(* Logix 5000 project; controller ERT303_BaseConfig vendor 1 type 14 code 226 rev 33.11; software revision 33.02 *)

TASK MainTask (continuous, watchdog 500 ms) : MainProgram
TASK SafetyTask (periodic, rate 20 ms, priority 10, watchdog 20 ms, safety) : SafetyProgram

MODULES
   Local : vendor 1 type 14 code 226 (5069 0, rev 33.11)
END_MODULES

TYPE _Blade :
STRUCT
   Raise : _sol_motion;
   Lower : _sol_motion;
END_STRUCT
END_TYPE

TYPE _clamp :
STRUCT
   Raise : _sol_motion;
   Lower : _sol_motion;
   Clamp : _sol_motion;
   Unclamp : _sol_motion;
END_STRUCT
END_TYPE

TYPE _Gantry :
STRUCT
   Adv_Z : _sol_motion;
   Ret_Z : _sol_motion;
   Adv_X : _sol_motion;
   Ret_X : _sol_motion;
   Grip : _sol_motion;
   Ungrip : _sol_motion;
   Adv_Y : _sol_motion;
   Ret_Y : _sol_motion;
END_STRUCT
END_TYPE

TYPE _modes :
STRUCT
   Auto : BOOL;   // Auto Mode
   Manual : BOOL;   // Manual Mode
   AutoCycle : BOOL;   // In Auto Cycle
END_STRUCT
END_TYPE

TYPE _motor :
STRUCT
   OkToMove : BOOL;   // Clear And OK To Move
   AutoCondition : BOOL;   // Auto Move Conditions Met
   Command : BOOL;   // Move Command
END_STRUCT
END_TYPE

TYPE _pusher :
STRUCT
   Adv : _sol_motion;   // Extend
   Ret : _sol_motion;   // Retract
END_STRUCT
END_TYPE

TYPE _sol_motion :
STRUCT
   OkToMove : BOOL;   // Clear And OK To Move
   AutoCondition : BOOL;   // Auto Move Conditions Met
   Command : BOOL;   // Move Command
   PosFdbk : BOOL;   // In Position Feedback
   Complete : BOOL;   // Motion Complete
   CompleteDelayTimer : TIMER;   // Motion Complete Delay Timer
   SlowFltTimer : TIMER;   // Slow Motion Fault Timer
   SlowFlt : BOOL;   // Slow Motion Fault
   SwitchFlt : BOOL;   // Switch Fault
END_STRUCT
END_TYPE

VAR_GLOBAL   (* controller tags *)
   AlarmSta1 : ALIAS FOR BOOL_OUT_17;   // ALARM AT STATION 1
   AlarmSta2 : ALIAS FOR BOOL_OUT_32;   // ALARM AT STATION 2
   BELT0 : ALIAS FOR BOOL_OUT_1;
   BELT1 : ALIAS FOR BOOL_OUT_2;
   BELT10 : ALIAS FOR BOOL_OUT_11;
   BELT11 : ALIAS FOR BOOL_OUT_12;
   BELT12 : ALIAS FOR BOOL_OUT_13;
   BELT13 : ALIAS FOR BOOL_OUT_14;
   BELT14 : ALIAS FOR BOOL_OUT_15;
   BELT2 : ALIAS FOR BOOL_OUT_3;
   BELT3 : ALIAS FOR BOOL_OUT_4;
   BELT4 : ALIAS FOR BOOL_OUT_5;
   BELT5 : ALIAS FOR BOOL_OUT_6;
   BELT6 : ALIAS FOR BOOL_OUT_7;
   BELT7 : ALIAS FOR BOOL_OUT_8;
   BELT8 : ALIAS FOR BOOL_OUT_9;
   BELT9 : ALIAS FOR BOOL_OUT_10;
   BELTWEIGHTSCALE : ALIAS FOR BOOL_OUT_16;
   BOOL_IN_1 : BOOL := 1;
   BOOL_IN_10 : BOOL;
   BOOL_IN_11 : BOOL;
   BOOL_IN_12 : BOOL;
   BOOL_IN_13 : BOOL;
   BOOL_IN_14 : BOOL;
   BOOL_IN_15 : BOOL;
   BOOL_IN_16 : BOOL;
   BOOL_IN_17 : BOOL;
   BOOL_IN_18 : BOOL;
   BOOL_IN_19 : BOOL;
   BOOL_IN_2 : BOOL;
   BOOL_IN_20 : BOOL;
   BOOL_IN_21 : BOOL;
   BOOL_IN_22 : BOOL;
   BOOL_IN_23 : BOOL;
   BOOL_IN_24 : BOOL;
   BOOL_IN_25 : BOOL;
   BOOL_IN_26 : BOOL;
   BOOL_IN_27 : BOOL;
   BOOL_IN_28 : BOOL;
   BOOL_IN_29 : BOOL;
   BOOL_IN_3 : BOOL := 1;
   BOOL_IN_30 : BOOL;
   BOOL_IN_31 : BOOL;
   BOOL_IN_32 : BOOL;
   BOOL_IN_33 : BOOL;
   BOOL_IN_34 : BOOL;
   BOOL_IN_35 : BOOL;
   BOOL_IN_36 : BOOL;
   BOOL_IN_4 : BOOL;
   BOOL_IN_5 : BOOL;
   BOOL_IN_6 : BOOL;
   BOOL_IN_7 : BOOL;
   BOOL_IN_8 : BOOL;
   BOOL_IN_9 : BOOL;
   BOOL_OUT_1 : BOOL;
   BOOL_OUT_10 : BOOL;
   BOOL_OUT_11 : BOOL;
   BOOL_OUT_12 : BOOL;
   BOOL_OUT_13 : BOOL;
   BOOL_OUT_14 : BOOL;
   BOOL_OUT_15 : BOOL;
   BOOL_OUT_16 : BOOL;
   BOOL_OUT_17 : BOOL := 1;
   BOOL_OUT_18 : BOOL;
   BOOL_OUT_19 : BOOL;
   BOOL_OUT_2 : BOOL;
   BOOL_OUT_20 : BOOL;
   BOOL_OUT_21 : BOOL;
   BOOL_OUT_22 : BOOL;
   BOOL_OUT_23 : BOOL;
   BOOL_OUT_24 : BOOL;
   BOOL_OUT_25 : BOOL;
   BOOL_OUT_26 : BOOL;
   BOOL_OUT_27 : BOOL;
   BOOL_OUT_28 : BOOL;
   BOOL_OUT_29 : BOOL := 1;
   BOOL_OUT_3 : BOOL;
   BOOL_OUT_30 : BOOL;
   BOOL_OUT_31 : BOOL := 1;
   BOOL_OUT_32 : BOOL := 1;
   BOOL_OUT_33 : BOOL;
   BOOL_OUT_34 : BOOL := 1;
   BOOL_OUT_35 : BOOL;
   BOOL_OUT_36 : BOOL;
   BOOL_OUT_37 : BOOL := 1;
   BOOL_OUT_38 : BOOL := 1;
   BOOL_OUT_39 : BOOL := 1;
   BOOL_OUT_4 : BOOL;
   BOOL_OUT_40 : BOOL := 1;
   BOOL_OUT_41 : BOOL;
   BOOL_OUT_42 : BOOL := 1;
   BOOL_OUT_43 : BOOL := 1;
   BOOL_OUT_44 : BOOL;
   BOOL_OUT_5 : BOOL;
   BOOL_OUT_6 : BOOL;
   BOOL_OUT_7 : BOOL;
   BOOL_OUT_8 : BOOL;
   BOOL_OUT_9 : BOOL;
   CURVEBELT0 : ALIAS FOR BOOL_OUT_18;
   CURVEBELT1 : ALIAS FOR BOOL_OUT_22;
   CURVEBELT2 : ALIAS FOR BOOL_OUT_19;
   CURVEBELT3 : ALIAS FOR BOOL_OUT_20;
   CURVEBELT4 : ALIAS FOR BOOL_OUT_21;
   DISPLAY0 : ALIAS FOR FLOAT_OUT_1;   // WEIGHT DISPLAY
   DISPLAY1 : ALIAS FOR INT_OUT_1;   // SHOWS TOTAL PARTS ON FRAGILE LINE
   DISPLAY2 : ALIAS FOR INT_OUT_2;   // SHOWS TOTAL NUMBER OF PARTS HANDLE BY SYSTEM
   EmergencyStop : ALIAS FOR BOOL_IN_1;   // EMERGENCY STOP BUTTON
   FactoryIOReset : ALIAS FOR BOOL_OUT_43;   // RESET BUTTON FOR WHOLE SYSTEM
   FLOAT_IN_1 : REAL;
   FLOAT_IN_10 : REAL;
   FLOAT_IN_11 : REAL;
   FLOAT_IN_12 : REAL;
   FLOAT_IN_2 : REAL;
   FLOAT_IN_3 : REAL;
   FLOAT_IN_4 : REAL;
   FLOAT_IN_5 : REAL;
   FLOAT_IN_6 : REAL;
   FLOAT_IN_7 : REAL;
   FLOAT_IN_8 : REAL;
   FLOAT_IN_9 : REAL;
   FLOAT_OUT_1 : REAL;
   FLOAT_OUT_10 : REAL;
   FLOAT_OUT_11 : REAL;
   FLOAT_OUT_12 : REAL;
   FLOAT_OUT_2 : REAL;
   FLOAT_OUT_3 : REAL;
   FLOAT_OUT_4 : REAL;
   FLOAT_OUT_5 : REAL;
   FLOAT_OUT_6 : REAL;
   FLOAT_OUT_7 : REAL;
   FLOAT_OUT_8 : REAL;
   FLOAT_OUT_9 : REAL;
   FRAGILESENSOR : ALIAS FOR BOOL_IN_5;   // SENSOR FOR FRAGILE PART COUNT AT STARTING OF FRAGILE LINE
   FRAGILESENSOR2 : ALIAS FOR BOOL_IN_23;   // SENSOR FOR FRAGILE PART COUNT AT ENDING OF FRAGILE LINE
   INT_IN_1 : DINT;
   INT_IN_10 : DINT;
   INT_IN_11 : DINT;
   INT_IN_12 : DINT;
   INT_IN_13 : DINT;
   INT_IN_14 : DINT;
   INT_IN_15 : DINT;
   INT_IN_16 : DINT;
   INT_IN_17 : DINT;
   INT_IN_18 : DINT;
   INT_IN_2 : DINT;
   INT_IN_3 : DINT;
   INT_IN_4 : DINT;
   INT_IN_5 : DINT;
   INT_IN_6 : DINT;
   INT_IN_7 : DINT;
   INT_IN_8 : DINT;
   INT_IN_9 : DINT;
   INT_OUT_1 : DINT := 3;
   INT_OUT_10 : DINT;
   INT_OUT_11 : DINT;
   INT_OUT_12 : DINT;
   INT_OUT_13 : DINT;
   INT_OUT_14 : DINT;
   INT_OUT_15 : DINT;
   INT_OUT_16 : DINT;
   INT_OUT_17 : DINT;
   INT_OUT_18 : DINT;
   INT_OUT_2 : DINT;
   INT_OUT_3 : DINT;
   INT_OUT_4 : DINT;
   INT_OUT_5 : DINT;
   INT_OUT_6 : DINT;
   INT_OUT_7 : DINT;
   INT_OUT_8 : DINT;
   INT_OUT_9 : DINT;
   PBRESET1 : ALIAS FOR BOOL_IN_16;   // RESET PB FOR STATION 1
   PBRESET2 : ALIAS FOR BOOL_IN_17;   // RESET PB OF STATION 2
   PIVOTARM0 : ALIAS FOR BOOL_OUT_23;   // MAIN PIVOT ARM
   PIVOTARM1 : ALIAS FOR BOOL_OUT_24;   // PIVOT ARM FOR SORTING OF BLUE PART
   PIVOTARM2 : ALIAS FOR BOOL_OUT_25;   // PIVOT ARM FOR SORTING OF GREEN PART
   PIVOTARMBELT0 : ALIAS FOR BOOL_OUT_26;
   PIVOTARMBELT1 : ALIAS FOR BOOL_OUT_27;
   PIVOTARMBELT2 : ALIAS FOR BOOL_OUT_28;
   SAFTEYDOOR : ALIAS FOR BOOL_IN_18;   // SAFTEYDOOR CONTROL
   STACKLTGREEN : ALIAS FOR BOOL_OUT_36;   // GREEN STACK LIGHT AT FRONT STATION
   STACKLTGREEN1 : ALIAS FOR BOOL_OUT_30;   // GREEN STACK LIGHT AT STATION 1
   STACKLTGREEN2 : ALIAS FOR BOOL_OUT_41;   // GREEN STACK LIGHT AT STATION 2
   STACKLTRED : ALIAS FOR BOOL_OUT_35;
   STACKLTRED1 : ALIAS FOR BOOL_OUT_29;   // RED STACK LIGHT AT STATION 1
   STACKLTRED2 : ALIAS FOR BOOL_OUT_40;   // RED STACK LIGHT AT STATION 2
   STACKLTYELLOW : ALIAS FOR BOOL_OUT_37;   // YELLOW STACK LIGHT AT FRONT
   STACKLTYELLOW1 : ALIAS FOR BOOL_OUT_31;   // YELLOW STACK LIGHT AT STATION 1
   STACKLTYELLOW2 : ALIAS FOR BOOL_OUT_42;   // YELLOW STACK LIGHT AT STATION 2
   STARTLT : ALIAS FOR BOOL_OUT_33;   // GREEN LIGHT OF START PB
   StartPB : ALIAS FOR BOOL_IN_2;   // START PUSH BUTTON
   STOPLT : ALIAS FOR BOOL_OUT_34;   // RED LIGHT OF STOP PB
   StopPB : ALIAS FOR BOOL_IN_3;   // STOP PUSH BUTTON
   VISION1A : ALIAS FOR BOOL_IN_6;
   VISION1B : ALIAS FOR BOOL_IN_7;
   VISION1C : ALIAS FOR BOOL_IN_8;
   VISION2A : ALIAS FOR BOOL_IN_9;
   VISION2B : ALIAS FOR BOOL_IN_10;
   VISION2C : ALIAS FOR BOOL_IN_11;
   VISION3A : ALIAS FOR BOOL_IN_12;
   VISION3B : ALIAS FOR BOOL_IN_13;
   VISION3C : ALIAS FOR BOOL_IN_14;
   VISION3D : ALIAS FOR BOOL_IN_15;
   VISION4A : ALIAS FOR BOOL_IN_19;
   VISION4B : ALIAS FOR BOOL_IN_20;
   VISION4C : ALIAS FOR BOOL_IN_21;
   VISION4D : ALIAS FOR BOOL_IN_22;
   WARNLTST1 : ALIAS FOR BOOL_OUT_39;   // WARN LIGHT AT FRAGILE PART PICKUP STATION
   WARNLTSTAIR : ALIAS FOR BOOL_OUT_38;   // WARN SIGNAL LIGHT AT STAIR
   WeightScale : ALIAS FOR FLOAT_IN_1;   // ACTUAL WEIGHT MEASURE AT WEIGHT SCALE
   WeightSensor : ALIAS FOR BOOL_IN_4;   // SENSOR AT WEIGHT SCALE
END_VAR

PROGRAM MainProgram   (* main routine MainRoutine *)
VAR
   ActualWeight : REAL;
   AllConveyorsRun : BOOL;   // All Conveyors present
   DelayTimer : TIMER := (PRE := 5000);   // DELAY OF 5 SECONDS AT WEIGHT BELT
   FRAGILEPARTS : COUNTER;
   FRAGILEPARTSTART : COUNTER := (ACC := 29, DN := 1);   // COUNTER OF FRAGILE PART AT START OF FRAGILE LINE
   FRAGILEPARTSTOP : COUNTER := (ACC := 26, DN := 1);   // COUNTER OF FRAGILE PART AT END OF FRAGILE LINE
   Partdelaycomplete : BOOL;   // PART DELAY COMPLETION
   TotalParts : COUNTER;   // TOTAL PARTS HANDLE BY SYSTEM
END_VAR

ROUTINE CONVEYOR_SYSTEM   (* ladder *)
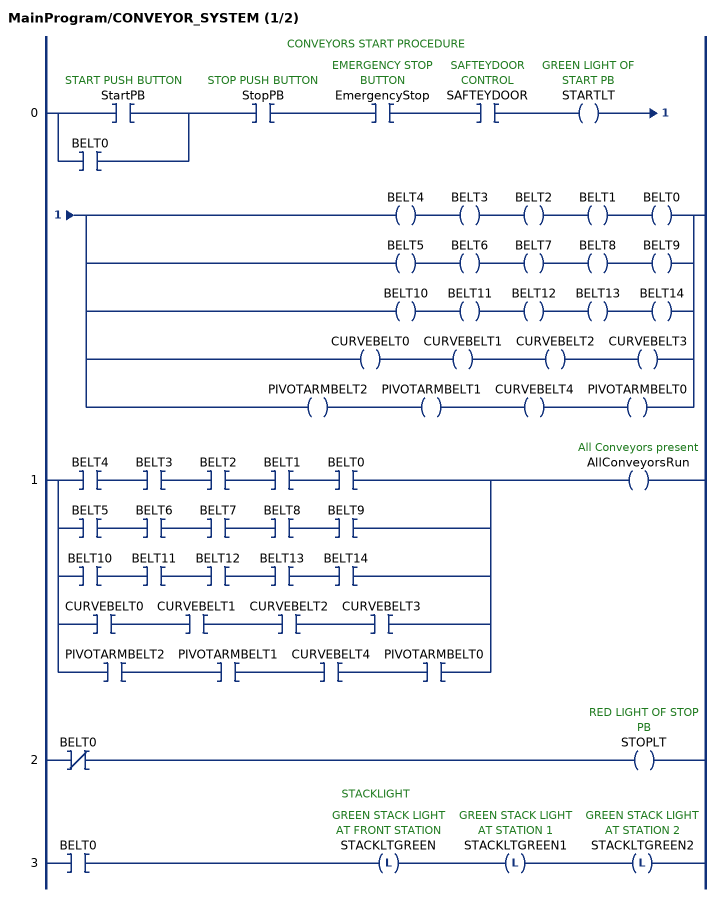
   // CONVEYORS START PROCEDURE
   0: [XIC(StartPB) ,XIC(BELT0) ]XIC(StopPB)XIC(EmergencyStop)XIC(SAFTEYDOOR)OTE(STARTLT)[OTE(BELT4) OTE(BELT3) OTE(BELT2) OTE(BELT1) OTE(BELT0) ,OTE(BELT5) OTE(BELT6) OTE(BELT7) OTE(BELT8) OTE(BELT9) ,OTE(BELT10) OTE(BELT11) OTE(BELT12) OTE(BELT13) OTE(BELT14) ,OTE(CURVEBELT0) OTE(CURVEBELT1) OTE(CURVEBELT2) OTE(CURVEBELT3) ,OTE(PIVOTARMBELT2) OTE(PIVOTARMBELT1) OTE(CURVEBELT4) OTE(PIVOTARMBELT0) ];
   1: [XIC(BELT4) XIC(BELT3) XIC(BELT2) XIC(BELT1) XIC(BELT0) ,XIC(BELT5) XIC(BELT6) XIC(BELT7) XIC(BELT8) XIC(BELT9) ,XIC(BELT10) XIC(BELT11) XIC(BELT12) XIC(BELT13) XIC(BELT14) ,XIC(CURVEBELT0) XIC(CURVEBELT1) XIC(CURVEBELT2) XIC(CURVEBELT3) ,XIC(PIVOTARMBELT2) XIC(PIVOTARMBELT1) XIC(CURVEBELT4) XIC(PIVOTARMBELT0) ]OTE(AllConveyorsRun);
   2: XIO(BELT0)OTE(STOPLT);
   // STACKLIGHT
   3: XIC(BELT0)OTL(STACKLTGREEN)OTL(STACKLTGREEN1)OTL(STACKLTGREEN2);
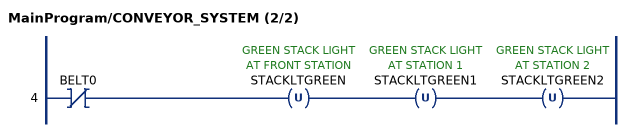
   4: XIO(BELT0)OTU(STACKLTGREEN)OTU(STACKLTGREEN1)OTU(STACKLTGREEN2);
END_ROUTINE

ROUTINE LIGHTING   (* ladder *)
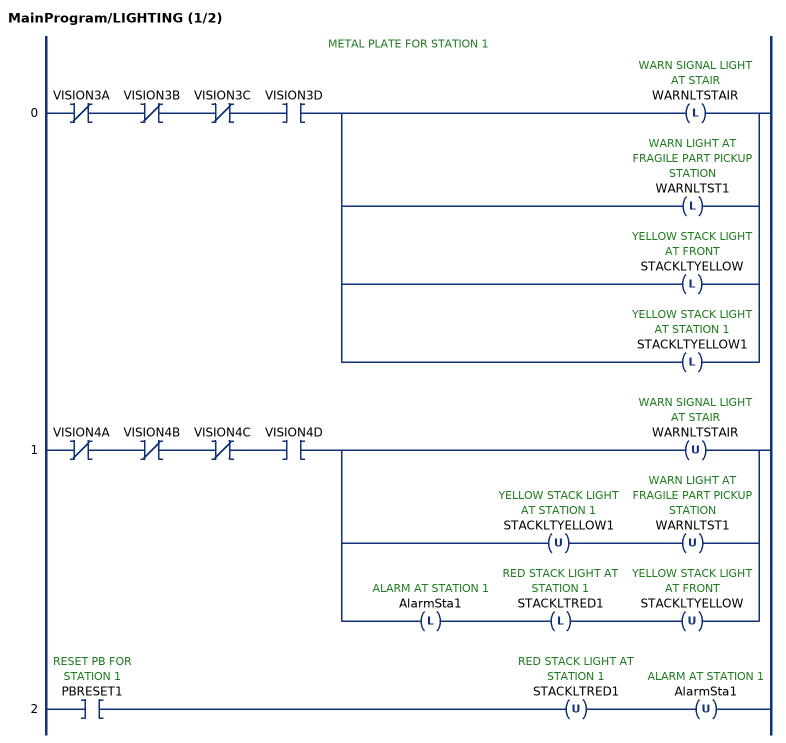
   // METAL PLATE FOR STATION 1
   0: XIO(VISION3A)XIO(VISION3B)XIO(VISION3C)XIC(VISION3D)[OTL(WARNLTSTAIR) ,OTL(WARNLTST1) ,OTL(STACKLTYELLOW) ,OTL(STACKLTYELLOW1) ];
   1: XIO(VISION4A)XIO(VISION4B)XIO(VISION4C)XIC(VISION4D)[OTU(WARNLTSTAIR) ,OTU(STACKLTYELLOW1) OTU(WARNLTST1) ,OTL(AlarmSta1) OTL(STACKLTRED1) OTU(STACKLTYELLOW) ];
   2: XIC(PBRESET1)OTU(STACKLTRED1)OTU(AlarmSta1);
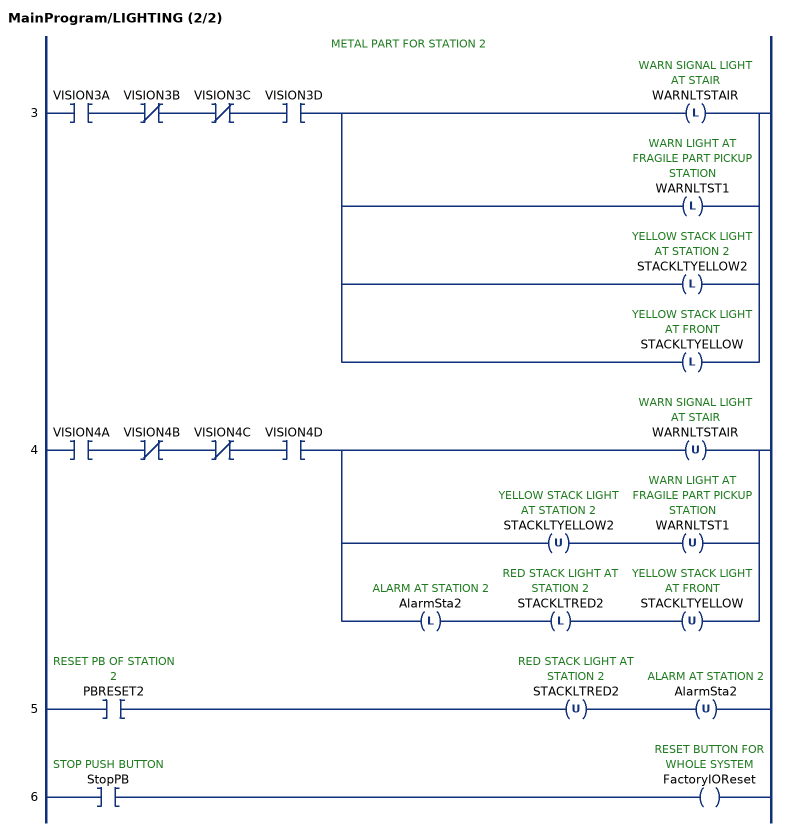
   // METAL PART FOR STATION 2
   3: XIC(VISION3A)XIO(VISION3B)XIO(VISION3C)XIC(VISION3D)[OTL(WARNLTSTAIR) ,OTL(WARNLTST1) ,OTL(STACKLTYELLOW2) ,OTL(STACKLTYELLOW) ];
   4: XIC(VISION4A)XIO(VISION4B)XIO(VISION4C)XIC(VISION4D)[OTU(WARNLTSTAIR) ,OTU(STACKLTYELLOW2) OTU(WARNLTST1) ,OTL(AlarmSta2) OTL(STACKLTRED2) OTU(STACKLTYELLOW) ];
   5: XIC(PBRESET2)OTU(STACKLTRED2)OTU(AlarmSta2);
   6: XIC(StopPB)OTE(FactoryIOReset);
END_ROUTINE

ROUTINE MainRoutine   (* ladder *)
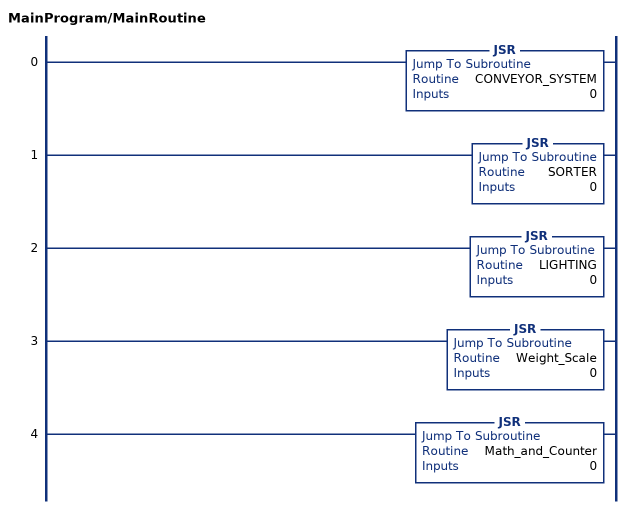
   0: JSR(CONVEYOR_SYSTEM,0);
   1: JSR(SORTER,0);
   2: JSR(LIGHTING,0);
   3: JSR(Weight_Scale,0);
   4: JSR(Math_and_Counter,0);
END_ROUTINE

ROUTINE Math_and_Counter   (* ladder *)
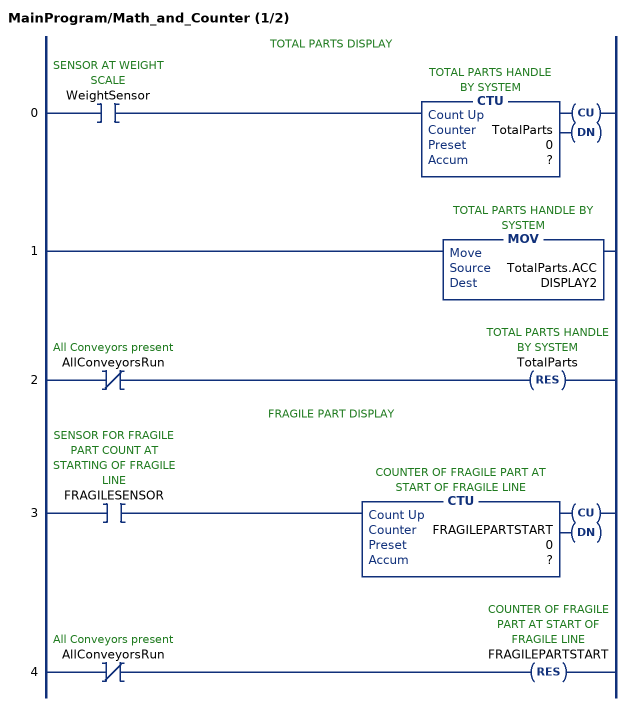
   // TOTAL PARTS DISPLAY
   0: XIC(WeightSensor)CTU(TotalParts,?,?);
   1: MOV(TotalParts.ACC,DISPLAY2);
   2: XIO(AllConveyorsRun)RES(TotalParts);
   // FRAGILE PART DISPLAY
   3: XIC(FRAGILESENSOR)CTU(FRAGILEPARTSTART,?,?);
   4: XIO(AllConveyorsRun)RES(FRAGILEPARTSTART);
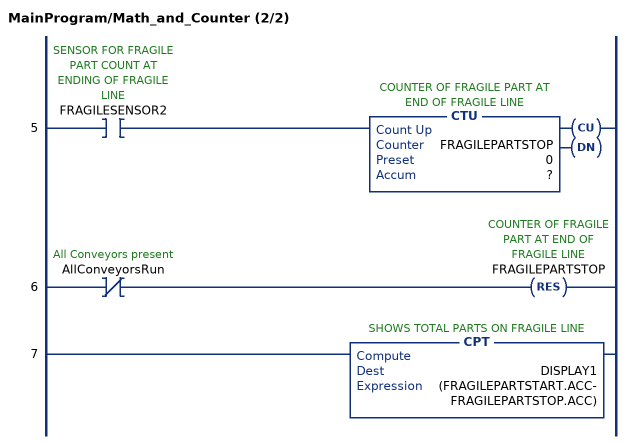
   5: XIC(FRAGILESENSOR2)CTU(FRAGILEPARTSTOP,?,?);
   6: XIO(AllConveyorsRun)RES(FRAGILEPARTSTOP);
   7: CPT(DISPLAY1,(FRAGILEPARTSTART.ACC-FRAGILEPARTSTOP.ACC));
END_ROUTINE

ROUTINE SORTER   (* ladder *)
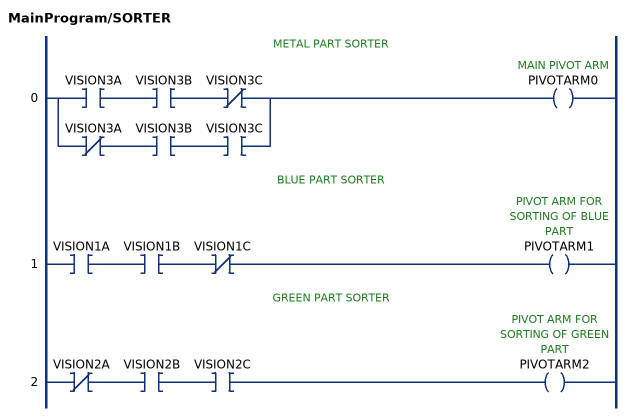
   // METAL PART SORTER
   0: [XIC(VISION3A) XIC(VISION3B) XIO(VISION3C) ,XIO(VISION3A) XIC(VISION3B) XIC(VISION3C) ]OTE(PIVOTARM0);
   // BLUE PART SORTER
   1: XIC(VISION1A)XIC(VISION1B)XIO(VISION1C)OTE(PIVOTARM1);
   // GREEN PART SORTER
   2: XIO(VISION2A)XIC(VISION2B)XIC(VISION2C)OTE(PIVOTARM2);
END_ROUTINE

ROUTINE Weight_Scale   (* ladder *)
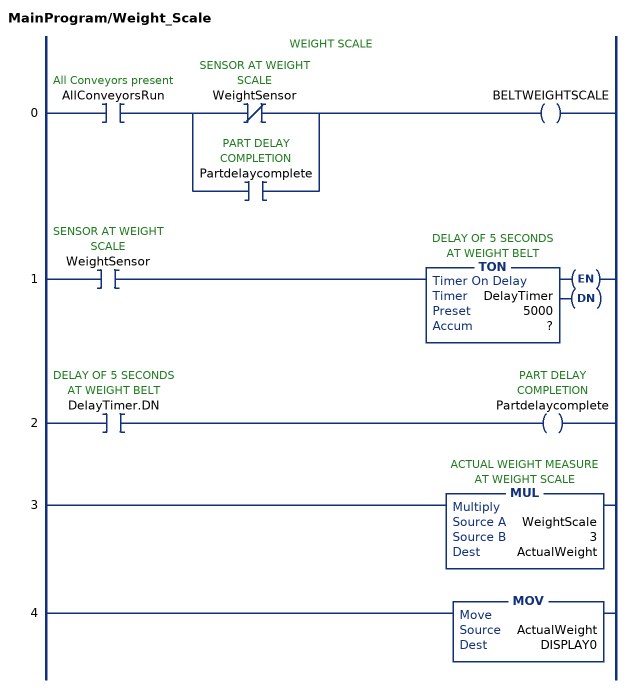
   // WEIGHT SCALE
   0: XIC(AllConveyorsRun)[XIO(WeightSensor) ,XIC(Partdelaycomplete) ]OTE(BELTWEIGHTSCALE);
   1: XIC(WeightSensor)TON(DelayTimer,?,?);
   2: XIC(DelayTimer.DN)OTE(Partdelaycomplete);
   3: MUL(WeightScale,3,ActualWeight);
   4: MOV(ActualWeight,DISPLAY0);
END_ROUTINE
END_PROGRAM

PROGRAM SafetyProgram   (* main routine MainRoutine, safety *)

ROUTINE MainRoutine   (* ladder *)
END_ROUTINE
END_PROGRAM
